Universal Robots PolyScope program: orange_Snap_buttom.urp

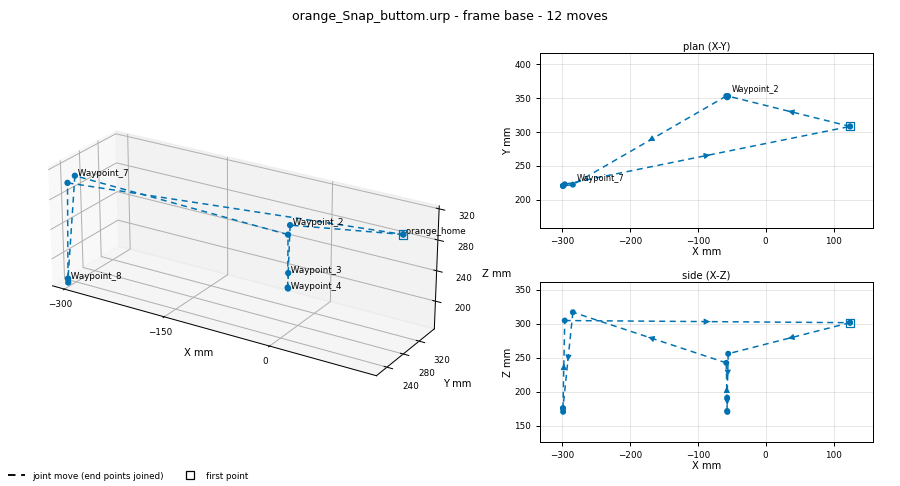
[picture p0: tool path of orange_Snap_buttom.urp in frame base, 12 of 12 moves have a stored position in this frame; points joined in program order, loops and branches not executed]
Program orange_Snap_buttom (installation=default directory=/programs/usbdisk/Zahra1/orangi createdIn=5.11.11.1010533 lastSavedIn=5.11.11.1010533 robotSerialNumber=20205300864)
Calibrated DH parameters: a=[-0.000166, -0.243494, -0.153108, 0.000057, -0.000123, 0]; d=[0.151897, -1.34267, 53.988124, -52.514559, 0.085283, 0.092193]; alpha=[1.572472, -0.003756, 0.002824, 1.570807, -1.572621, 0]; deltaTheta=[0, 0.020704, 7.033215, -0.770746, 0.000004, 0]
Robot Program (runOnlyOnce=true)
  MoveJ speed 60 deg/s, acceleration 80 deg/s^2 (useActiveTCP=true) feature=Base
    Waypoint orange_home: TCP in base x=124.286 y=308.277 z=301.462 mm, rx=2.2499 ry=-2.1846 rz=-0.0963 rad; joints [-269.66, -91.226, -90.279, -86.086, 92.69, 808.818] deg
    URCap Gripper (Robotiq_Grippers, Robotiq Inc.) dataModel(position=33.72549019607843, force=94.0, speed=40.0, positionInDouble=33.72549019607843, forceInDouble=94.0, speedInDouble=40.0, slaveIds=[9], blocking=true, robotCompliant=false)
    Waypoint Waypoint_2: TCP in base x=-55.16 y=352.892 z=255.74 mm, rx=-2.2135 ry=2.22 rz=-0.0593 rad; joints [-239.474, -99.575, -91.614, -80.72, 89.137, 840.833] deg
    Waypoint Waypoint_3: TCP in base x=-56.716 y=352.167 z=190.96 mm, rx=2.205 ry=-2.2253 rz=0.0496 rad; joints [-239.455, -104.766, -103.703, -63.306, 90.041, 841.237] deg
    Waypoint Waypoint_4: TCP in base x=-56.377 y=351.572 z=170.042 mm, rx=2.205 ry=-2.2253 rz=0.0495 rad; joints [-239.46, -107.267, -106.852, -57.651, 90.033, 841.244] deg
    URCap Gripper (Robotiq_Grippers, Robotiq Inc.) dataModel(position=62.431372549019606, force=94.0, speed=40.0, positionInDouble=62.431372549019606, forceInDouble=94.0, speedInDouble=40.0, slaveIds=[9], blocking=true, robotCompliant=false)
    Waypoint Waypoint_5: TCP in base x=-56.705 y=351.113 z=171.372 mm, rx=2.196 ry=-2.2376 rz=0.0498 rad; joints [-239.336, -106.977, -106.841, -57.927, 89.911, 841.92] deg
    Waypoint Waypoint_6: TCP in base x=-58.006 y=353.03 z=242.265 mm, rx=2.1961 ry=-2.2376 rz=0.0498 rad; joints [-239.285, -100.495, -94.285, -76.964, 89.913, 841.924] deg
    Waypoint Waypoint_7: TCP in base x=-283.957 y=222.508 z=316.84 mm, rx=-2.0739 ry=2.2618 rz=0.0906 rad; joints [-195.43, -97.918, -78.233, -93.061, 84.717, 889.587] deg
    Waypoint Waypoint_8: TCP in base x=-298.551 y=220.821 z=175.467 mm, rx=-2.1863 ry=2.2191 rz=-0.0532 rad; joints [-195.886, -109.947, -101.023, -61.362, 89.67, 885.141] deg
    Waypoint Waypoint_9: TCP in base x=-298.323 y=220.777 z=170.211 mm, rx=-2.1863 ry=2.2191 rz=-0.0532 rad; joints [-195.891, -110.562, -101.78, -59.989, 89.669, 885.138] deg
    URCap Gripper (Robotiq_Grippers, Robotiq Inc.) dataModel(position=25.098039215686274, force=94.0, speed=40.0, positionInDouble=25.098039215686274, forceInDouble=94.0, speedInDouble=40.0, slaveIds=[9], blocking=true, robotCompliant=false)
    Waypoint Waypoint_8: TCP in base x=-298.551 y=220.821 z=175.467 mm, rx=-2.1863 ry=2.2191 rz=-0.0532 rad; joints [-195.886, -109.947, -101.023, -61.362, 89.67, 885.141] deg
    Waypoint Waypoint_10: TCP in base x=-295.942 y=223.084 z=304.62 mm, rx=-2.167 ry=2.2272 rz=0.0621 rad; joints [-195.653, -100.602, -78.397, -89.884, 87.174, 885.985] deg
    Waypoint orange_home: TCP in base x=124.286 y=308.277 z=301.462 mm, rx=2.2499 ry=-2.1846 rz=-0.0963 rad; joints [-269.66, -91.226, -90.279, -86.086, 92.69, 808.818] deg
